FUNCTION_BLOCK FB_PositionStatePMPS EXTENDS FB_PositionStatePMPS_Base
(*
    Hooks up a position state to an arbiter and an FFO
        Use BeamParameterTransitionManager to manage transition requests between states
        Hook up to the inputs/outputs of the state function block
        Raises FFO if beam parameters are worse than required for current state
*)
VAR_IN_OUT
    fbArbiter: FB_Arbiter;
    fbFFHWO: FB_HardwareFFOutput;
END_VAR
VAR
    bptm: BeamParameterTransitionManager;
    ffBeamParamsOk: FB_FastFault;
    bFFOxOk: BOOL;
END_VAR

Exec();

ACTION HandleBPTM:
bptm(fbArbiter:=fbArbiter,
     i_TransitionAssertionID:=nTransitionAssertionID,
     i_stTransitionAssertion:=stTransitionBeam,
     i_nRequestedAssertionID:=stStateReq.nRequestAssertionID,
     i_stRequestedAssertion:=stStateReq.stBeamParams,
     i_xMoving:=bDoingTransition,
     i_xDoneMoving:=NOT bDoingTransition,
     stCurrentBeamParameters:=PMPS_GVL.stCurrentBeamParameters,
     q_xTransitionAuthorized=>bTransitionAuthorized);
END_ACTION

ACTION HandleFFO:
// If the beam parameters are wrong, it is a fault! This encompasses all arbiter-related errors.
// Get state will point to Unknown/No beam if we are out of state bounds or in motion
// Otherwise we'll have the current state's beam parameters
IF stBeamNeeded.nRate <= 0 THEN
    bFFOxOk := FALSE;
ELSE
    bFFOxOk := F_SafeBPCompare(PMPS_GVL.stCurrentBeamParameters, stBeamNeeded);
END_IF
ffBeamParamsOk(
    i_xOK:=bFFOxOk,
    i_DevName:=stMotionStage.sName,
    i_Desc:='Beam parameter mismatch',
    io_fbFFHWO:=fbFFHWO);
END_ACTION

END_FUNCTION_BLOCK

(* stored: Version 1.1.0.1, ProductVersion 3.1.4022.18
   POU FB_PositionStatePMPS: Id {7e0e3094-8a3d-4636-a390-eb10e10412f0}, SpecialFunc None
   Action HandleBPTM: Id {15e95ede-ce74-498f-962a-8707e856078c}
   Action HandleFFO: Id {6b3afb71-b9c2-4718-aacf-85bf75e65e9c} *)
